LIN {X 0,Y 80.87,Z 798.949,A -85,B 0,C 180,E1 4987.72,E2 4987.72} C_VEL
LIN {X 0,Y 77.511,Z 800.568,A -85,B 0,C 180,E1 4982.778,E2 4982.778} C_VEL
LIN {X 0,Y 74.215,Z 804.27,A -85,B 0,C 180,E1 4966.959,E2 4966.959} C_VEL
LIN {X 0,Y 75.459,Z 805.862,A -85,B 0,C 180,E1 4953.038,E2 4953.038} C_VEL
LIN {X 0,Y 75.99,Z 806.028,A -85,B 0,C 180,E1 4949.467,E2 4949.467} C_VEL
LIN {X 0,Y 74.209,Z 804.782,A -85,B 0,C 180,E1 4936.759,E2 4936.759} C_VEL
LIN {X 0,Y 76.212,Z 801.556,A -85,B 0,C 180,E1 4920.961,E2 4920.961} C_VEL
LIN {X 0,Y 83.236,Z 796.479,A -85,B 0,C 180,E1 4906.789,E2 4906.789} C_VEL
LIN {X 0,Y 94.398,Z 789.488,A -85,B 0,C 180,E1 4895.358,E2 4895.358} C_VEL
LIN {X 0,Y 107.739,Z 780.951,A -85,B 0,C 180,E1 4887.014,E2 4887.014} C_VEL
LIN {X 0,Y 122.056,Z 770.983,A -85,B 0,C 180,E1 4880.958,E2 4880.958} C_VEL
LIN {X 0,Y 136.611,Z 759.652,A -85,B 0,C 180,E1 4876.511,E2 4876.511} C_VEL
LIN {X 0,Y 150.961,Z 747,A -85,B 0,C 180,E1 4873.195,E2 4873.195} C_VEL
LIN {X 0,Y 165.296,Z 732.474,A -85,B 0,C 180,E1 4870.605,E2 4870.605} C_VEL
LIN {X 0,Y 178.339,Z 717.175,A -85,B 0,C 180,E1 4868.706,E2 4868.706} C_VEL
LIN {X 0,Y 190.774,Z 700.081,A -85,B 0,C 180,E1 4867.225,E2 4867.225} C_VEL
LIN {X 0,Y 201.627,Z 682.331,A -85,B 0,C 180,E1 4866.151,E2 4866.151} C_VEL
LIN {X 0,Y 211.381,Z 662.929,A -85,B 0,C 180,E1 4865.337,E2 4865.337} C_VEL
LIN {X 0,Y 219.258,Z 643.158,A -85,B 0,C 180,E1 4864.725,E2 4864.725} C_VEL
LIN {X 0,Y 225.387,Z 622.689,A -85,B 0,C 180,E1 4864.227,E2 4864.227} C_VEL
LIN {X 0,Y 229.672,Z 601.778,A -85,B 0,C 180,E1 4863.811,E2 4863.811} C_VEL
LIN {X 0,Y 238.268,Z 530.43,A -85,B 0,C 180,E1 4862.645,E2 4862.645} C_VEL
LIN {X 0,Y 237.776,Z 527.887,A -85,B 0,C 180,E1 4860.24,E2 4860.24} C_VEL
LIN {X 0,Y 237.596,Z 526.381,A -85,B 0,C 180,E1 4858.07,E2 4858.07} C_VEL
LIN {X 0,Y 237.865,Z 526.25,A -85,B 0,C 180,E1 4853.967,E2 4853.967} C_VEL
LIN {X 0,Y 238.211,Z 526.899,A -85,B 0,C 180,E1 4852.402,E2 4852.402} C_VEL
LIN {X 0,Y 238.456,Z 528.071,A -85,B 0,C 180,E1 4851.324,E2 4851.324} C_VEL
LIN {X 0,Y 231.321,Z 589.425,A -85,B 0,C 180,E1 4850.247,E2 4850.247} C_VEL
LIN {X 0,Y 228.042,Z 608.919,A -85,B 0,C 180,E1 4849.701,E2 4849.701} C_VEL
LIN {X 0,Y 223.305,Z 627.563,A -85,B 0,C 180,E1 4849.015,E2 4849.015} C_VEL
LIN {X 0,Y 217.088,Z 645.659,A -85,B 0,C 180,E1 4848.153,E2 4848.153} C_VEL
LIN {X 0,Y 208.731,Z 664.585,A -85,B 0,C 180,E1 4846.988,E2 4846.988} C_VEL
LIN {X 0,Y 198.839,Z 682.549,A -85,B 0,C 180,E1 4845.556,E2 4845.556} C_VEL
LIN {X 0,Y 187.897,Z 698.953,A -85,B 0,C 180,E1 4843.836,E2 4843.836} C_VEL
LIN {X 0,Y 175.842,Z 714.135,A -85,B 0,C 180,E1 4841.724,E2 4841.724} C_VEL
LIN {X 0,Y 162.701,Z 728.173,A -85,B 0,C 180,E1 4839.079,E2 4839.079} C_VEL
LIN {X 0,Y 149.063,Z 740.606,A -85,B 0,C 180,E1 4835.812,E2 4835.812} C_VEL
LIN {X 0,Y 135.111,Z 751.51,A -85,B 0,C 180,E1 4831.716,E2 4831.716} C_VEL
LIN {X 0,Y 120.926,Z 761.042,A -85,B 0,C 180,E1 4826.358,E2 4826.358} C_VEL
LIN {X 0,Y 107.001,Z 769.093,A -85,B 0,C 180,E1 4819.19,E2 4819.19} C_VEL
LIN {X 0,Y 94.79,Z 775.203,A -85,B 0,C 180,E1 4810.047,E2 4810.047} C_VEL
LIN {X 0,Y 85.286,Z 779.428,A -85,B 0,C 180,E1 4798.728,E2 4798.728} C_VEL
LIN {X 0,Y 79.196,Z 781.917,A -85,B 0,C 180,E1 4785.374,E2 4785.374} C_VEL
LIN {X 0,Y 77.022,Z 782.778,A -85,B 0,C 180,E1 4770.744,E2 4770.744} C_VEL
LIN {X 0,Y 78.595,Z 782.144,A -85,B 0,C 180,E1 4756.763,E2 4756.763} C_VEL
LIN {X 0,Y 84.097,Z 779.929,A -85,B 0,C 180,E1 4743.142,E2 4743.142} C_VEL
LIN {X 0,Y 93.116,Z 776.003,A -85,B 0,C 180,E1 4731.481,E2 4731.481} C_VEL
LIN {X 0,Y 104.314,Z 770.552,A -85,B 0,C 180,E1 4722.436,E2 4722.436} C_VEL
LIN {X 0,Y 117.401,Z 763.276,A -85,B 0,C 180,E1 4715.158,E2 4715.158} C_VEL
LIN {X 0,Y 131.069,Z 754.49,A -85,B 0,C 180,E1 4709.586,E2 4709.586} C_VEL
LIN {X 0,Y 145.656,Z 743.569,A -85,B 0,C 180,E1 4705.03,E2 4705.03} C_VEL
LIN {X 0,Y 159.184,Z 731.747,A -85,B 0,C 180,E1 4701.631,E2 4701.631} C_VEL
LIN {X 0,Y 172.242,Z 718.44,A -85,B 0,C 180,E1 4698.884,E2 4698.884} C_VEL
LIN {X 0,Y 184.101,Z 704.311,A -85,B 0,C 180,E1 4696.73,E2 4696.73} C_VEL
LIN {X 0,Y 195.07,Z 688.928,A -85,B 0,C 180,E1 4694.95,E2 4694.95} C_VEL
LIN {X 0,Y 205.1,Z 672.108,A -85,B 0,C 180,E1 4693.461,E2 4693.461} C_VEL
LIN {X 0,Y 213.82,Z 654.238,A -85,B 0,C 180,E1 4692.234,E2 4692.234} C_VEL
LIN {X 0,Y 220.959,Z 635.839,A -85,B 0,C 180,E1 4691.251,E2 4691.251} C_VEL
LIN {X 0,Y 226.74,Z 615.995,A -85,B 0,C 180,E1 4690.436,E2 4690.436} C_VEL
LIN {X 0,Y 230.757,Z 595.786,A -85,B 0,C 180,E1 4689.81,E2 4689.81} C_VEL
LIN {X 0,Y 236.026,Z 551.57,A -85,B 0,C 180,E1 4688.94,E2 4688.94} C_VEL
LIN {X 0,Y 238.75,Z 528.075,A -85,B 0,C 180,E1 4688.563,E2 4688.563} C_VEL
LIN {X 0,Y 238.273,Z 526.572,A -85,B 0,C 180,E1 4686.506,E2 4686.506} C_VEL
LIN {X 0,Y 237.888,Z 526.562,A -85,B 0,C 180,E1 4682.168,E2 4682.168} C_VEL
LIN {X 0,Y 238.215,Z 528.774,A -85,B 0,C 180,E1 4678.918,E2 4678.918} C_VEL
LIN {X 0,Y 238.522,Z 530.833,A -85,B 0,C 180,E1 4677.356,E2 4677.356} C_VEL
LIN {X 0,Y 229.693,Z 603.415,A -85,B 0,C 180,E1 4676.168,E2 4676.168} C_VEL
LIN {X 0,Y 225.268,Z 624.242,A -85,B 0,C 180,E1 4675.75,E2 4675.75} C_VEL
LIN {X 0,Y 219.212,Z 644.095,A -85,B 0,C 180,E1 4675.261,E2 4675.261} C_VEL
LIN {X 0,Y 211.383,Z 663.553,A -85,B 0,C 180,E1 4674.655,E2 4674.655} C_VEL
LIN {X 0,Y 202.115,Z 681.945,A -85,B 0,C 180,E1 4673.885,E2 4673.885} C_VEL
LIN {X 0,Y 190.896,Z 700.299,A -85,B 0,C 180,E1 4672.779,E2 4672.779} C_VEL
LIN {X 0,Y 178.447,Z 717.368,A -85,B 0,C 180,E1 4671.299,E2 4671.299} C_VEL
LIN {X 0,Y 164.832,Z 733.27,A -85,B 0,C 180,E1 4669.311,E2 4669.311} C_VEL
LIN {X 0,Y 150.054,Z 748.089,A -85,B 0,C 180,E1 4666.61,E2 4666.61} C_VEL
LIN {X 0,Y 134.86,Z 761.302,A -85,B 0,C 180,E1 4663.016,E2 4663.016} C_VEL
LIN {X 0,Y 119.586,Z 772.97,A -85,B 0,C 180,E1 4658.131,E2 4658.131} C_VEL
LIN {X 0,Y 104.755,Z 783.066,A -85,B 0,C 180,E1 4651.412,E2 4651.412} C_VEL
LIN {X 0,Y 91.293,Z 791.543,A -85,B 0,C 180,E1 4642.049,E2 4642.049} C_VEL
LIN {X 0,Y 81.046,Z 798.03,A -85,B 0,C 180,E1 4629.904,E2 4629.904} C_VEL
LIN {X 0,Y 77.511,Z 800.568,A -85,B 0,C 180,E1 4622.778,E2 4622.778} C_VEL
LIN {X 0,Y 74.757,Z 801.989,A -85,B 0,C 180,E1 4617.407,E2 4617.407} C_VEL
LIN {X 0,Y 68.448,Z 803.712,A -85,B 0,C 180,E1 4605.965,E2 4605.965} C_VEL
LIN {X 0,Y 66.797,Z 804.343,A -85,B 0,C 180,E1 4598.037,E2 4598.037} C_VEL
LIN {X 0,Y 66.981,Z 804.481,A -85,B 0,C 180,E1 4595.654,E2 4595.654} C_VEL
LIN {X 0,Y 67.99,Z 804.819,A -85,B 0,C 180,E1 4589.63,E2 4589.63} C_VEL
LIN {X 0,Y 66.248,Z 803.424,A -85,B 0,C 180,E1 4574.237,E2 4574.237} C_VEL
LIN {X 0,Y 69.077,Z 800.295,A -85,B 0,C 180,E1 4557.619,E2 4557.619} C_VEL
LIN {X 0,Y 77.372,Z 795.212,A -85,B 0,C 180,E1 4542.559,E2 4542.559} C_VEL
LIN {X 0,Y 89.824,Z 788.216,A -85,B 0,C 180,E1 4531.009,E2 4531.009} C_VEL
LIN {X 0,Y 104.215,Z 779.674,A -85,B 0,C 180,E1 4522.924,E2 4522.924} C_VEL
LIN {X 0,Y 119.332,Z 769.699,A -85,B 0,C 180,E1 4517.223,E2 4517.223} C_VEL
LIN {X 0,Y 134.489,Z 758.36,A -85,B 0,C 180,E1 4513.12,E2 4513.12} C_VEL
LIN {X 0,Y 149.29,Z 745.693,A -85,B 0,C 180,E1 4510.102,E2 4510.102} C_VEL
LIN {X 0,Y 163.502,Z 731.675,A -85,B 0,C 180,E1 4507.843,E2 4507.843} C_VEL
LIN {X 0,Y 176.979,Z 716.205,A -85,B 0,C 180,E1 4506.12,E2 4506.12} C_VEL
LIN {X 0,Y 189.635,Z 699.109,A -85,B 0,C 180,E1 4504.808,E2 4504.808} C_VEL
LIN {X 0,Y 200.918,Z 680.865,A -85,B 0,C 180,E1 4503.846,E2 4503.846} C_VEL
LIN {X 0,Y 210.287,Z 662.45,A -85,B 0,C 180,E1 4503.175,E2 4503.175} C_VEL
LIN {X 0,Y 218.195,Z 642.955,A -85,B 0,C 180,E1 4502.643,E2 4502.643} C_VEL
LIN {X 0,Y 224.532,Z 622.209,A -85,B 0,C 180,E1 4502.192,E2 4502.192} C_VEL
LIN {X 0,Y 228.935,Z 601.111,A -85,B 0,C 180,E1 4501.809,E2 4501.809} C_VEL
LIN {X 0,Y 236.861,Z 536.432,A -85,B 0,C 180,E1 4500.801,E2 4500.801} C_VEL
LIN {X 0,Y 236.592,Z 534.278,A -85,B 0,C 180,E1 4497.82,E2 4497.82} C_VEL
LIN {X 0,Y 236.945,Z 534.241,A -85,B 0,C 180,E1 4493.701,E2 4493.701} C_VEL
LIN {X 0,Y 237.048,Z 534.547,A -85,B 0,C 180,E1 4493.152,E2 4493.152} C_VEL
LIN {X 0,Y 230.283,Z 591.262,A -85,B 0,C 180,E1 4492.187,E2 4492.187} C_VEL
LIN {X 0,Y 226.761,Z 611.086,A -85,B 0,C 180,E1 4491.649,E2 4491.649} C_VEL
LIN {X 0,Y 221.706,Z 630.042,A -85,B 0,C 180,E1 4490.977,E2 4490.977} C_VEL
LIN {X 0,Y 215.141,Z 648.362,A -85,B 0,C 180,E1 4490.141,E2 4490.141} C_VEL
LIN {X 0,Y 206.72,Z 666.747,A -85,B 0,C 180,E1 4489.064,E2 4489.064} C_VEL
LIN {X 0,Y 196.939,Z 684.033,A -85,B 0,C 180,E1 4487.766,E2 4487.766} C_VEL
LIN {X 0,Y 185.854,Z 700.262,A -85,B 0,C 180,E1 4486.174,E2 4486.174} C_VEL
LIN {X 0,Y 173.527,Z 715.411,A -85,B 0,C 180,E1 4484.201,E2 4484.201} C_VEL
LIN {X 0,Y 160.047,Z 729.424,A -85,B 0,C 180,E1 4481.724,E2 4481.724} C_VEL
LIN {X 0,Y 145.999,Z 741.842,A -85,B 0,C 180,E1 4478.647,E2 4478.647} C_VEL
LIN {X 0,Y 131.542,Z 752.736,A -85,B 0,C 180,E1 4474.756,E2 4474.756} C_VEL
LIN {X 0,Y 116.962,Z 762.108,A -85,B 0,C 180,E1 4469.699,E2 4469.699} C_VEL
LIN {X 0,Y 102.702,Z 769.932,A -85,B 0,C 180,E1 4462.967,E2 4462.967} C_VEL
LIN {X 0,Y 89.463,Z 776.145,A -85,B 0,C 180,E1 4453.861,E2 4453.861} C_VEL
LIN {X 0,Y 78.868,Z 780.452,A -85,B 0,C 180,E1 4442.171,E2 4442.171} C_VEL
LIN {X 0,Y 71.832,Z 783.018,A -85,B 0,C 180,E1 4427.832,E2 4427.832} C_VEL
LIN {X 0,Y 69.156,Z 783.937,A -85,B 0,C 180,E1 4412.486,E2 4412.486} C_VEL
LIN {X 0,Y 70.527,Z 783.466,A -85,B 0,C 180,E1 4396.89,E2 4396.89} C_VEL
LIN {X 0,Y 76.303,Z 781.422,A -85,B 0,C 180,E1 4381.854,E2 4381.854} C_VEL
LIN {X 0,Y 85.91,Z 777.677,A -85,B 0,C 180,E1 4369.328,E2 4369.328} C_VEL
LIN {X 0,Y 98.445,Z 772.088,A -85,B 0,C 180,E1 4359.478,E2 4359.478} C_VEL
LIN {X 0,Y 112.253,Z 764.919,A -85,B 0,C 180,E1 4352.204,E2 4352.204} C_VEL
LIN {X 0,Y 126.523,Z 756.253,A -85,B 0,C 180,E1 4346.752,E2 4346.752} C_VEL
LIN {X 0,Y 140.772,Z 746.14,A -85,B 0,C 180,E1 4342.584,E2 4342.584} C_VEL
LIN {X 0,Y 154.677,Z 734.619,A -85,B 0,C 180,E1 4339.311,E2 4339.311} C_VEL
LIN {X 0,Y 168.049,Z 721.668,A -85,B 0,C 180,E1 4336.687,E2 4336.687} C_VEL
LIN {X 0,Y 180.762,Z 707.191,A -85,B 0,C 180,E1 4334.543,E2 4334.543} C_VEL
LIN {X 0,Y 192.724,Z 690.993,A -85,B 0,C 180,E1 4332.756,E2 4332.756} C_VEL
LIN {X 0,Y 202.946,Z 674.402,A -85,B 0,C 180,E1 4331.366,E2 4331.366} C_VEL
LIN {X 0,Y 211.824,Z 656.824,A -85,B 0,C 180,E1 4330.219,E2 4330.219} C_VEL
LIN {X 0,Y 219.327,Z 638.171,A -85,B 0,C 180,E1 4329.269,E2 4329.269} C_VEL
LIN {X 0,Y 225.338,Z 618.422,A -85,B 0,C 180,E1 4328.491,E2 4328.491} C_VEL
LIN {X 0,Y 229.599,Z 598.14,A -85,B 0,C 180,E1 4327.882,E2 4327.882} C_VEL
LIN {X 0,Y 234.631,Z 557.443,A -85,B 0,C 180,E1 4327.085,E2 4327.085} C_VEL
LIN {X 0,Y 237.333,Z 534.597,A -85,B 0,C 180,E1 4326.714,E2 4326.714} C_VEL
LIN {X 0,Y 236.89,Z 534.461,A -85,B 0,C 180,E1 4322.42,E2 4322.42} C_VEL
LIN {X 0,Y 237.097,Z 536.385,A -85,B 0,C 180,E1 4319.517,E2 4319.517} C_VEL
LIN {X 0,Y 237.127,Z 536.857,A -85,B 0,C 180,E1 4319.187,E2 4319.187} C_VEL
LIN {X 0,Y 228.983,Z 602.568,A -85,B 0,C 180,E1 4318.174,E2 4318.174} C_VEL
LIN {X 0,Y 224.534,Z 623.283,A -85,B 0,C 180,E1 4317.795,E2 4317.795} C_VEL
LIN {X 0,Y 218.444,Z 643.068,A -85,B 0,C 180,E1 4317.363,E2 4317.363} C_VEL
LIN {X 0,Y 210.782,Z 661.997,A -85,B 0,C 180,E1 4316.851,E2 4316.851} C_VEL
LIN {X 0,Y 200.92,Z 681.371,A -85,B 0,C 180,E1 4316.147,E2 4316.147} C_VEL
LIN {X 0,Y 189.637,Z 699.509,A -85,B 0,C 180,E1 4315.184,E2 4315.184} C_VEL
LIN {X 0,Y 176.981,Z 716.533,A -85,B 0,C 180,E1 4313.873,E2 4313.873} C_VEL
LIN {X 0,Y 163.027,Z 732.455,A -85,B 0,C 180,E1 4312.081,E2 4312.081} C_VEL
LIN {X 0,Y 148.356,Z 746.799,A -85,B 0,C 180,E1 4309.72,E2 4309.72} C_VEL
LIN {X 0,Y 132.674,Z 760.024,A -85,B 0,C 180,E1 4306.444,E2 4306.444} C_VEL
LIN {X 0,Y 116.739,Z 771.695,A -85,B 0,C 180,E1 4301.93,E2 4301.93} C_VEL
LIN {X 0,Y 101.029,Z 781.796,A -85,B 0,C 180,E1 4295.571,E2 4295.571} C_VEL
LIN {X 0,Y 86.409,Z 790.275,A -85,B 0,C 180,E1 4286.419,E2 4286.419} C_VEL
LIN {X 0,Y 74.612,Z 796.891,A -85,B 0,C 180,E1 4273.646,E2 4273.646} C_VEL
LIN {X 0,Y 67.665,Z 801.488,A -85,B 0,C 180,E1 4257.556,E2 4257.556} C_VEL
LIN {X 0,Y 66.421,Z 804.095,A -85,B 0,C 180,E1 4240.407,E2 4240.407} C_VEL
LIN {X 0,Y 66.981,Z 804.481,A -85,B 0,C 180,E1 4235.654,E2 4235.654} C_VEL
LIN {X 0,Y 66.693,Z 804.571,A -85,B 0,C 180,E1 4232.598,E2 4232.598} C_VEL
LIN {X 0,Y 64.66,Z 804.284,A -85,B 0,C 180,E1 4228.461,E2 4228.461} C_VEL
LIN {X 0,Y 58.75,Z 802.884,A -85,B 0,C 180,E1 4218.157,E2 4218.157} C_VEL
LIN {X 0,Y 58.309,Z 802.507,A -85,B 0,C 180,E1 4215.107,E2 4215.107} C_VEL
LIN {X 0,Y 61.542,Z 799.446,A -85,B 0,C 180,E1 4195.346,E2 4195.346} C_VEL
LIN {X 0,Y 70.802,Z 794.549,A -85,B 0,C 180,E1 4179.042,E2 4179.042} C_VEL
LIN {X 0,Y 83.558,Z 788.148,A -85,B 0,C 180,E1 4167.692,E2 4167.692} C_VEL
LIN {X 0,Y 99.129,Z 779.667,A -85,B 0,C 180,E1 4159.441,E2 4159.441} C_VEL
LIN {X 0,Y 115.328,Z 769.658,A -85,B 0,C 180,E1 4153.838,E2 4153.838} C_VEL
LIN {X 0,Y 130.975,Z 758.559,A -85,B 0,C 180,E1 4150.019,E2 4150.019} C_VEL
LIN {X 0,Y 147.104,Z 745.276,A -85,B 0,C 180,E1 4147.101,E2 4147.101} C_VEL
LIN {X 0,Y 162.096,Z 730.871,A -85,B 0,C 180,E1 4145.026,E2 4145.026} C_VEL
LIN {X 0,Y 176.293,Z 714.854,A -85,B 0,C 180,E1 4143.469,E2 4143.469} C_VEL
LIN {X 0,Y 189.126,Z 697.707,A -85,B 0,C 180,E1 4142.343,E2 4142.343} C_VEL
LIN {X 0,Y 200.04,Z 680.284,A -85,B 0,C 180,E1 4141.56,E2 4141.56} C_VEL
LIN {X 0,Y 209.496,Z 661.945,A -85,B 0,C 180,E1 4140.993,E2 4140.993} C_VEL
LIN {X 0,Y 217.523,Z 642.437,A -85,B 0,C 180,E1 4140.537,E2 4140.537} C_VEL
LIN {X 0,Y 223.931,Z 621.816,A -85,B 0,C 180,E1 4140.145,E2 4140.145} C_VEL
LIN {X 0,Y 228.431,Z 600.737,A -85,B 0,C 180,E1 4139.801,E2 4139.801} C_VEL
LIN {X 0,Y 235.632,Z 543.029,A -85,B 0,C 180,E1 4138.966,E2 4138.966} C_VEL
LIN {X 0,Y 235.593,Z 542.128,A -85,B 0,C 180,E1 4137.324,E2 4137.324} C_VEL
LIN {X 0,Y 235.733,Z 542.122,A -85,B 0,C 180,E1 4134.985,E2 4134.985} C_VEL
LIN {X 0,Y 229.443,Z 593.572,A -85,B 0,C 180,E1 4134.131,E2 4134.131} C_VEL
LIN {X 0,Y 225.559,Z 614.046,A -85,B 0,C 180,E1 4133.593,E2 4133.593} C_VEL
LIN {X 0,Y 220.134,Z 633.241,A -85,B 0,C 180,E1 4132.937,E2 4132.937} C_VEL
LIN {X 0,Y 212.981,Z 652.126,A -85,B 0,C 180,E1 4132.109,E2 4132.109} C_VEL
LIN {X 0,Y 204.421,Z 669.941,A -85,B 0,C 180,E1 4131.112,E2 4131.112} C_VEL
LIN {X 0,Y 194.523,Z 686.751,A -85,B 0,C 180,E1 4129.916,E2 4129.916} C_VEL
LIN {X 0,Y 183.19,Z 702.748,A -85,B 0,C 180,E1 4128.433,E2 4128.433} C_VEL
LIN {X 0,Y 170.616,Z 717.665,A -85,B 0,C 180,E1 4126.601,E2 4126.601} C_VEL
LIN {X 0,Y 157.746,Z 730.671,A -85,B 0,C 180,E1 4124.453,E2 4124.453} C_VEL
LIN {X 0,Y 143.306,Z 743.076,A -85,B 0,C 180,E1 4121.596,E2 4121.596} C_VEL
LIN {X 0,Y 128.363,Z 753.961,A -85,B 0,C 180,E1 4117.957,E2 4117.957} C_VEL
LIN {X 0,Y 113.169,Z 763.326,A -85,B 0,C 180,E1 4113.166,E2 4113.166} C_VEL
LIN {X 0,Y 97.751,Z 771.333,A -85,B 0,C 180,E1 4106.471,E2 4106.471} C_VEL
LIN {X 0,Y 83.271,Z 777.616,A -85,B 0,C 180,E1 4097.09,E2 4097.09} C_VEL
LIN {X 0,Y 71.46,Z 781.937,A -85,B 0,C 180,E1 4084.355,E2 4084.355} C_VEL
LIN {X 0,Y 63.8,Z 784.403,A -85,B 0,C 180,E1 4068.266,E2 4068.266} C_VEL
LIN {X 0,Y 61.2,Z 785.2,A -85,B 0,C 180,E1 4050,E2 4050} C_VEL
LIN {X 0,Y 63.781,Z 784.429,A -85,B 0,C 180,E1 4031.729,E2 4031.729} C_VEL
LIN {X 0,Y 71.262,Z 782.046,A -85,B 0,C 180,E1 4015.861,E2 4015.861} C_VEL
LIN {X 0,Y 82.576,Z 777.942,A -85,B 0,C 180,E1 4003.408,E2 4003.408} C_VEL
LIN {X 0,Y 95.818,Z 772.302,A -85,B 0,C 180,E1 3994.479,E2 3994.479} C_VEL
LIN {X 0,Y 109.848,Z 765.261,A -85,B 0,C 180,E1 3988.007,E2 3988.007} C_VEL
LIN {X 0,Y 124.866,Z 756.375,A -85,B 0,C 180,E1 3982.952,E2 3982.952} C_VEL
LIN {X 0,Y 139.694,Z 746.022,A -85,B 0,C 180,E1 3979.133,E2 3979.133} C_VEL
LIN {X 0,Y 154.055,Z 734.233,A -85,B 0,C 180,E1 3976.152,E2 3976.152} C_VEL
LIN {X 0,Y 167.795,Z 720.972,A -85,B 0,C 180,E1 3973.77,E2 3973.77} C_VEL
LIN {X 0,Y 180.342,Z 706.72,A -85,B 0,C 180,E1 3971.895,E2 3971.895} C_VEL
LIN {X 0,Y 191.484,Z 691.818,A -85,B 0,C 180,E1 3970.405,E2 3970.405} C_VEL
LIN {X 0,Y 201.999,Z 674.988,A -85,B 0,C 180,E1 3969.114,E2 3969.114} C_VEL
LIN {X 0,Y 211.047,Z 657.306,A -85,B 0,C 180,E1 3968.057,E2 3968.057} C_VEL
LIN {X 0,Y 218.915,Z 637.859,A -85,B 0,C 180,E1 3967.149,E2 3967.149} C_VEL
LIN {X 0,Y 224.94,Z 617.986,A -85,B 0,C 180,E1 3966.432,E2 3966.432} C_VEL
LIN {X 0,Y 229.184,Z 597.547,A -85,B 0,C 180,E1 3965.866,E2 3965.866} C_VEL
LIN {X 0,Y 234.66,Z 553.561,A -85,B 0,C 180,E1 3965.077,E2 3965.077} C_VEL
LIN {X 0,Y 236.022,Z 542.248,A -85,B 0,C 180,E1 3964.901,E2 3964.901} C_VEL
LIN {X 0,Y 235.911,Z 542.576,A -85,B 0,C 180,E1 3961.944,E2 3961.944} C_VEL
LIN {X 0,Y 235.906,Z 543.467,A -85,B 0,C 180,E1 3961.03,E2 3961.03} C_VEL
LIN {X 0,Y 228.524,Z 601.888,A -85,B 0,C 180,E1 3960.186,E2 3960.186} C_VEL
LIN {X 0,Y 224.052,Z 622.449,A -85,B 0,C 180,E1 3959.849,E2 3959.849} C_VEL
LIN {X 0,Y 217.921,Z 642.174,A -85,B 0,C 180,E1 3959.475,E2 3959.475} C_VEL
LIN {X 0,Y 209.994,Z 661.529,A -85,B 0,C 180,E1 3959.027,E2 3959.027} C_VEL
LIN {X 0,Y 200.538,Z 679.92,A -85,B 0,C 180,E1 3958.464,E2 3958.464} C_VEL
LIN {X 0,Y 189.127,Z 698.131,A -85,B 0,C 180,E1 3957.649,E2 3957.649} C_VEL
LIN {X 0,Y 176.294,Z 715.199,A -85,B 0,C 180,E1 3956.523,E2 3956.523} C_VEL
LIN {X 0,Y 162.585,Z 730.642,A -85,B 0,C 180,E1 3955.025,E2 3955.025} C_VEL
LIN {X 0,Y 147.106,Z 745.507,A -85,B 0,C 180,E1 3952.891,E2 3952.891} C_VEL
LIN {X 0,Y 130.978,Z 758.744,A -85,B 0,C 180,E1 3949.975,E2 3949.975} C_VEL
LIN {X 0,Y 114.43,Z 770.421,A -85,B 0,C 180,E1 3945.897,E2 3945.897} C_VEL
LIN {X 0,Y 97.874,Z 780.525,A -85,B 0,C 180,E1 3940.022,E2 3940.022} C_VEL
LIN {X 0,Y 82.085,Z 789.006,A -85,B 0,C 180,E1 3931.282,E2 3931.282} C_VEL
LIN {X 0,Y 69.092,Z 795.5,A -85,B 0,C 180,E1 3918.806,E2 3918.806} C_VEL
LIN {X 0,Y 60.631,Z 800.105,A -85,B 0,C 180,E1 3901.849,E2 3901.849} C_VEL
LIN {X 0,Y 58.387,Z 802.851,A -85,B 0,C 180,E1 3881.858,E2 3881.858} C_VEL
LIN {X 0,Y 59.99,Z 803.61,A -85,B 0,C 180,E1 3869.92,E2 3869.92} C_VEL
LIN {X 0,Y 58.309,Z 802.507,A -85,B 0,C 180,E1 3855.107,E2 3855.107} C_VEL
LIN {X 0,Y 57.755,Z 801.514,A -85,B 0,C 180,E1 3847.524,E2 3847.524} C_VEL
LIN {X 0,Y 57.592,Z 797.296,A -85,B 0,C 180,E1 3826.102,E2 3826.102} C_VEL
LIN {X 0,Y 59.976,Z 795.854,A -85,B 0,C 180,E1 3820.775,E2 3820.775} C_VEL
LIN {X 0,Y 72.988,Z 790.122,A -85,B 0,C 180,E1 3807.075,E2 3807.075} C_VEL
LIN {X 0,Y 88.363,Z 782.767,A -85,B 0,C 180,E1 3798.11,E2 3798.11} C_VEL
LIN {X 0,Y 104.879,Z 773.742,A -85,B 0,C 180,E1 3792.106,E2 3792.106} C_VEL
LIN {X 0,Y 121.175,Z 763.407,A -85,B 0,C 180,E1 3788.053,E2 3788.053} C_VEL
LIN {X 0,Y 137.53,Z 751.311,A -85,B 0,C 180,E1 3785.139,E2 3785.139} C_VEL
LIN {X 0,Y 153.668,Z 737.323,A -85,B 0,C 180,E1 3782.983,E2 3782.983} C_VEL
LIN {X 0,Y 168.442,Z 722.251,A -85,B 0,C 180,E1 3781.454,E2 3781.454} C_VEL
LIN {X 0,Y 181.972,Z 705.964,A -85,B 0,C 180,E1 3780.349,E2 3780.349} C_VEL
LIN {X 0,Y 193.973,Z 688.764,A -85,B 0,C 180,E1 3779.563,E2 3779.563} C_VEL
LIN {X 0,Y 204.496,Z 670.555,A -85,B 0,C 180,E1 3779.006,E2 3779.006} C_VEL
LIN {X 0,Y 213.528,Z 651.227,A -85,B 0,C 180,E1 3778.59,E2 3778.59} C_VEL
LIN {X 0,Y 220.816,Z 631.121,A -85,B 0,C 180,E1 3778.242,E2 3778.242} C_VEL
LIN {X 0,Y 226.297,Z 610.268,A -85,B 0,C 180,E1 3777.927,E2 3777.927} C_VEL
LIN {X 0,Y 229.862,Z 588.948,A -85,B 0,C 180,E1 3777.629,E2 3777.629} C_VEL
LIN {X 0,Y 234.62,Z 550.029,A -85,B 0,C 180,E1 3777.068,E2 3777.068} C_VEL
LIN {X 0,Y 234.603,Z 550.172,A -85,B 0,C 180,E1 3776.831,E2 3776.831} C_VEL
LIN {X 0,Y 228.774,Z 596.534,A -85,B 0,C 180,E1 3776.072,E2 3776.072} C_VEL
LIN {X 0,Y 224.789,Z 616.292,A -85,B 0,C 180,E1 3775.574,E2 3775.574} C_VEL
LIN {X 0,Y 219.306,Z 634.998,A -85,B 0,C 180,E1 3774.974,E2 3774.974} C_VEL
LIN {X 0,Y 212.044,Z 653.683,A -85,B 0,C 180,E1 3774.214,E2 3774.214} C_VEL
LIN {X 0,Y 202.871,Z 672.256,A -85,B 0,C 180,E1 3773.253,E2 3773.253} C_VEL
LIN {X 0,Y 192.291,Z 689.613,A -85,B 0,C 180,E1 3772.104,E2 3772.104} C_VEL
LIN {X 0,Y 180.343,Z 705.825,A -85,B 0,C 180,E1 3770.695,E2 3770.695} C_VEL
LIN {X 0,Y 167.071,Z 720.899,A -85,B 0,C 180,E1 3768.948,E2 3768.948} C_VEL
LIN {X 0,Y 152.678,Z 734.658,A -85,B 0,C 180,E1 3766.749,E2 3766.749} C_VEL
LIN {X 0,Y 137.345,Z 747.003,A -85,B 0,C 180,E1 3763.929,E2 3763.929} C_VEL
LIN {X 0,Y 121.154,Z 757.938,A -85,B 0,C 180,E1 3760.185,E2 3760.185} C_VEL
LIN {X 0,Y 105.121,Z 766.97,A -85,B 0,C 180,E1 3755.258,E2 3755.258} C_VEL
LIN {X 0,Y 89.249,Z 774.383,A -85,B 0,C 180,E1 3748.365,E2 3748.365} C_VEL
LIN {X 0,Y 74.638,Z 780.002,A -85,B 0,C 180,E1 3738.604,E2 3738.604} C_VEL
LIN {X 0,Y 62.804,Z 783.772,A -85,B 0,C 180,E1 3724.968,E2 3724.968} C_VEL
LIN {X 0,Y 55.242,Z 785.846,A -85,B 0,C 180,E1 3706.833,E2 3706.833} C_VEL
LIN {X 0,Y 53.351,Z 786.348,A -85,B 0,C 180,E1 3686.777,E2 3686.777} C_VEL
LIN {X 0,Y 56.942,Z 785.467,A -85,B 0,C 180,E1 3667.276,E2 3667.276} C_VEL
LIN {X 0,Y 65.952,Z 782.941,A -85,B 0,C 180,E1 3650.453,E2 3650.453} C_VEL
LIN {X 0,Y 78.749,Z 778.667,A -85,B 0,C 180,E1 3638.078,E2 3638.078} C_VEL
LIN {X 0,Y 93.957,Z 772.498,A -85,B 0,C 180,E1 3629.24,E2 3629.24} C_VEL
LIN {X 0,Y 109.988,Z 764.604,A -85,B 0,C 180,E1 3623.011,E2 3623.011} C_VEL
LIN {X 0,Y 126.173,Z 754.999,A -85,B 0,C 180,E1 3618.481,E2 3618.481} C_VEL
LIN {X 0,Y 141.882,Z 743.858,A -85,B 0,C 180,E1 3615.11,E2 3615.11} C_VEL
LIN {X 0,Y 156.749,Z 731.349,A -85,B 0,C 180,E1 3612.526,E2 3612.526} C_VEL
LIN {X 0,Y 171.051,Z 717.058,A -85,B 0,C 180,E1 3610.441,E2 3610.441} C_VEL
LIN {X 0,Y 184.125,Z 701.487,A -85,B 0,C 180,E1 3608.778,E2 3608.778} C_VEL
LIN {X 0,Y 195.624,Z 685.09,A -85,B 0,C 180,E1 3607.464,E2 3607.464} C_VEL
LIN {X 0,Y 205.693,Z 667.69,A -85,B 0,C 180,E1 3606.389,E2 3606.389} C_VEL
LIN {X 0,Y 214.444,Z 648.925,A -85,B 0,C 180,E1 3605.481,E2 3605.481} C_VEL
LIN {X 0,Y 221.561,Z 629.164,A -85,B 0,C 180,E1 3604.733,E2 3604.733} C_VEL
LIN {X 0,Y 226.833,Z 608.925,A -85,B 0,C 180,E1 3604.135,E2 3604.135} C_VEL
LIN {X 0,Y 230.244,Z 588.417,A -85,B 0,C 180,E1 3603.668,E2 3603.668} C_VEL
LIN {X 0,Y 234.909,Z 550.241,A -85,B 0,C 180,E1 3603.05,E2 3603.05} C_VEL
LIN {X 0,Y 234.874,Z 550.537,A -85,B 0,C 180,E1 3602.885,E2 3602.885} C_VEL
LIN {X 0,Y 228.383,Z 601.024,A -85,B 0,C 180,E1 3602.206,E2 3602.206} C_VEL
LIN {X 0,Y 223.867,Z 621.585,A -85,B 0,C 180,E1 3601.909,E2 3601.909} C_VEL
LIN {X 0,Y 217.741,Z 641.16,A -85,B 0,C 180,E1 3601.596,E2 3601.596} C_VEL
LIN {X 0,Y 210.013,Z 659.968,A -85,B 0,C 180,E1 3601.24,E2 3601.24} C_VEL
LIN {X 0,Y 200.347,Z 678.704,A -85,B 0,C 180,E1 3600.778,E2 3600.778} C_VEL
LIN {X 0,Y 188.968,Z 696.743,A -85,B 0,C 180,E1 3600.12,E2 3600.12} C_VEL
LIN {X 0,Y 175.988,Z 713.859,A -85,B 0,C 180,E1 3599.186,E2 3599.186} C_VEL
LIN {X 0,Y 161.571,Z 729.855,A -85,B 0,C 180,E1 3597.873,E2 3597.873} C_VEL
LIN {X 0,Y 146.112,Z 744.389,A -85,B 0,C 180,E1 3596.077,E2 3596.077} C_VEL
LIN {X 0,Y 129.791,Z 757.463,A -85,B 0,C 180,E1 3593.583,E2 3593.583} C_VEL
LIN {X 0,Y 112.691,Z 769.146,A -85,B 0,C 180,E1 3590.004,E2 3590.004} C_VEL
LIN {X 0,Y 95.347,Z 779.255,A -85,B 0,C 180,E1 3584.738,E2 3584.738} C_VEL
LIN {X 0,Y 78.415,Z 787.738,A -85,B 0,C 180,E1 3576.64,E2 3576.64} C_VEL
LIN {X 0,Y 63.911,Z 794.235,A -85,B 0,C 180,E1 3564.438,E2 3564.438} C_VEL
LIN {X 0,Y 53.764,Z 798.845,A -85,B 0,C 180,E1 3546.519,E2 3546.519} C_VEL
LIN {X 0,Y 50.391,Z 801.627,A -85,B 0,C 180,E1 3523.538,E2 3523.538} C_VEL
LIN {X 0,Y 51.916,Z 802.384,A -85,B 0,C 180,E1 3510,E2 3510} C_VEL
LIN {X 0,Y 50.587,Z 800.922,A -85,B 0,C 180,E1 3489.16,E2 3489.16} C_VEL
LIN {X 0,Y 56.209,Z 797.564,A -85,B 0,C 180,E1 3467.473,E2 3467.473} C_VEL
LIN {X 0,Y 59.976,Z 795.854,A -85,B 0,C 180,E1 3460.775,E2 3460.775} C_VEL
LIN {X 0,Y 63.488,Z 793.944,A -85,B 0,C 180,E1 3454.597,E2 3454.597} C_VEL
LIN {X 0,Y 73.141,Z 787.653,A -85,B 0,C 180,E1 3439.522,E2 3439.522} C_VEL
LIN {X 0,Y 77.807,Z 785.332,A -85,B 0,C 180,E1 3436.368,E2 3436.368} C_VEL
LIN {X 0,Y 94.429,Z 777.363,A -85,B 0,C 180,E1 3430.037,E2 3430.037} C_VEL
LIN {X 0,Y 111.547,Z 767.711,A -85,B 0,C 180,E1 3425.775,E2 3425.775} C_VEL
LIN {X 0,Y 129.127,Z 755.981,A -85,B 0,C 180,E1 3422.751,E2 3422.751} C_VEL
LIN {X 0,Y 145.985,Z 742.671,A -85,B 0,C 180,E1 3420.653,E2 3420.653} C_VEL
LIN {X 0,Y 161.488,Z 728.226,A -85,B 0,C 180,E1 3419.199,E2 3419.199} C_VEL
LIN {X 0,Y 175.559,Z 712.766,A -85,B 0,C 180,E1 3418.173,E2 3418.173} C_VEL
LIN {X 0,Y 188.154,Z 696.372,A -85,B 0,C 180,E1 3417.452,E2 3417.452} C_VEL
LIN {X 0,Y 199.249,Z 679.077,A -85,B 0,C 180,E1 3416.947,E2 3416.947} C_VEL
LIN {X 0,Y 208.833,Z 660.918,A -85,B 0,C 180,E1 3416.594,E2 3416.594} C_VEL
LIN {X 0,Y 212.676,Z 652.363,A -85,B 0,C 180,E1 3416.453,E2 3416.453} C_VEL
LIN {X 0,Y 204.053,Z 670.181,A -85,B 0,C 180,E1 3415.652,E2 3415.652} C_VEL
LIN {X 0,Y 193.664,Z 687.596,A -85,B 0,C 180,E1 3414.667,E2 3414.667} C_VEL
LIN {X 0,Y 182.141,Z 703.588,A -85,B 0,C 180,E1 3413.496,E2 3413.496} C_VEL
LIN {X 0,Y 169.105,Z 718.73,A -85,B 0,C 180,E1 3412.031,E2 3412.031} C_VEL
LIN {X 0,Y 155.214,Z 732.323,A -85,B 0,C 180,E1 3410.254,E2 3410.254} C_VEL
LIN {X 0,Y 140.061,Z 744.825,A -85,B 0,C 180,E1 3407.954,E2 3407.954} C_VEL
LIN {X 0,Y 124.215,Z 755.806,A -85,B 0,C 180,E1 3404.995,E2 3404.995} C_VEL
LIN {X 0,Y 107.843,Z 765.272,A -85,B 0,C 180,E1 3401.025,E2 3401.025} C_VEL
LIN {X 0,Y 91.236,Z 773.187,A -85,B 0,C 180,E1 3395.447,E2 3395.447} C_VEL
LIN {X 0,Y 75.702,Z 779.207,A -85,B 0,C 180,E1 3387.702,E2 3387.702} C_VEL
LIN {X 0,Y 61.349,Z 783.693,A -85,B 0,C 180,E1 3375.814,E2 3375.814} C_VEL
LIN {X 0,Y 50.55,Z 786.423,A -85,B 0,C 180,E1 3358.34,E2 3358.34} C_VEL
LIN {X 0,Y 45.608,Z 787.501,A -85,B 0,C 180,E1 3336.293,E2 3336.293} C_VEL
LIN {X 0,Y 47.165,Z 787.194,A -85,B 0,C 180,E1 3312.736,E2 3312.736} C_VEL
LIN {X 0,Y 55.349,Z 785.326,A -85,B 0,C 180,E1 3292.108,E2 3292.108} C_VEL
LIN {X 0,Y 67.439,Z 782.004,A -85,B 0,C 180,E1 3278.209,E2 3278.209} C_VEL
LIN {X 0,Y 82.847,Z 776.709,A -85,B 0,C 180,E1 3268.239,E2 3268.239} C_VEL
LIN {X 0,Y 98.957,Z 769.858,A -85,B 0,C 180,E1 3261.638,E2 3261.638} C_VEL
LIN {X 0,Y 115.928,Z 761.002,A -85,B 0,C 180,E1 3256.799,E2 3256.799} C_VEL
LIN {X 0,Y 132.531,Z 750.496,A -85,B 0,C 180,E1 3253.296,E2 3253.296} C_VEL
LIN {X 0,Y 147.58,Z 739.153,A -85,B 0,C 180,E1 3250.78,E2 3250.78} C_VEL
LIN {X 0,Y 162.832,Z 725.464,A -85,B 0,C 180,E1 3248.668,E2 3248.668} C_VEL
LIN {X 0,Y 176.794,Z 710.501,A -85,B 0,C 180,E1 3247.017,E2 3247.017} C_VEL
LIN {X 0,Y 189.401,Z 694.329,A -85,B 0,C 180,E1 3245.691,E2 3245.691} C_VEL
LIN {X 0,Y 200.614,Z 676.933,A -85,B 0,C 180,E1 3244.607,E2 3244.607} C_VEL
LIN {X 0,Y 209.954,Z 659.194,A -85,B 0,C 180,E1 3243.74,E2 3243.74} C_VEL
LIN {X 0,Y 212.304,Z 653.923,A -85,B 0,C 180,E1 3243.519,E2 3243.519} C_VEL
LIN {X 0,Y 203.282,Z 672.394,A -85,B 0,C 180,E1 3243.202,E2 3243.202} C_VEL
LIN {X 0,Y 192.691,Z 690.076,A -85,B 0,C 180,E1 3242.762,E2 3242.762} C_VEL
LIN {X 0,Y 180.67,Z 706.774,A -85,B 0,C 180,E1 3242.133,E2 3242.133} C_VEL
LIN {X 0,Y 167.642,Z 722.073,A -85,B 0,C 180,E1 3241.274,E2 3241.274} C_VEL
LIN {X 0,Y 152.974,Z 736.714,A -85,B 0,C 180,E1 3240.04,E2 3240.04} C_VEL
LIN {X 0,Y 137.036,Z 750.232,A -85,B 0,C 180,E1 3238.303,E2 3238.303} C_VEL
LIN {X 0,Y 120.293,Z 762.301,A -85,B 0,C 180,E1 3235.86,E2 3235.86} C_VEL
LIN {X 0,Y 102.399,Z 773.217,A -85,B 0,C 180,E1 3232.144,E2 3232.144} C_VEL
LIN {X 0,Y 84.326,Z 782.486,A -85,B 0,C 180,E1 3226.471,E2 3226.471} C_VEL
LIN {X 0,Y 67.139,Z 789.96,A -85,B 0,C 180,E1 3217.413,E2 3217.413} C_VEL
LIN {X 0,Y 52.493,Z 795.592,A -85,B 0,C 180,E1 3202.449,E2 3202.449} C_VEL
LIN {X 0,Y 43.546,Z 799.345,A -85,B 0,C 180,E1 3178.827,E2 3178.827} C_VEL
LIN {X 0,Y 43.371,Z 801.043,A -85,B 0,C 180,E1 3152.642,E2 3152.642} C_VEL
LIN {X 0,Y 43.798,Z 801.151,A -85,B 0,C 180,E1 3150,E2 3150} C_VEL
LIN {X 0,Y 42.989,Z 799.656,A -85,B 0,C 180,E1 3125.099,E2 3125.099} C_VEL
LIN {X 0,Y 50.39,Z 796.299,A -85,B 0,C 180,E1 3101.063,E2 3101.063} C_VEL
LIN {X 0,Y 63.995,Z 791.093,A -85,B 0,C 180,E1 3084.949,E2 3084.949} C_VEL
LIN {X 0,Y 77.807,Z 785.332,A -85,B 0,C 180,E1 3076.368,E2 3076.368} C_VEL
LIN {X 0,Y 83.405,Z 782.539,A -85,B 0,C 180,E1 3073.103,E2 3073.103} C_VEL
LIN {X 0,Y 96.694,Z 774.657,A -85,B 0,C 180,E1 3064.844,E2 3064.844} C_VEL
LIN {X 0,Y 102.777,Z 771.132,A -85,B 0,C 180,E1 3062.957,E2 3062.957} C_VEL
LIN {X 0,Y 119.98,Z 760.841,A -85,B 0,C 180,E1 3060.179,E2 3060.179} C_VEL
LIN {X 0,Y 137.042,Z 748.732,A -85,B 0,C 180,E1 3058.227,E2 3058.227} C_VEL
LIN {X 0,Y 153.203,Z 735.16,A -85,B 0,C 180,E1 3056.867,E2 3056.867} C_VEL
LIN {X 0,Y 168.403,Z 720.049,A -85,B 0,C 180,E1 3055.895,E2 3055.895} C_VEL
LIN {X 0,Y 176.106,Z 711.289,A -85,B 0,C 180,E1 3055.477,E2 3055.477} C_VEL
LIN {X 0,Y 161.85,Z 726.387,A -85,B 0,C 180,E1 3054.033,E2 3054.033} C_VEL
LIN {X 0,Y 146.33,Z 740.113,A -85,B 0,C 180,E1 3052.197,E2 3052.197} C_VEL
LIN {X 0,Y 130.009,Z 752.149,A -85,B 0,C 180,E1 3049.86,E2 3049.86} C_VEL
LIN {X 0,Y 112.984,Z 762.559,A -85,B 0,C 180,E1 3046.761,E2 3046.761} C_VEL
LIN {X 0,Y 95.439,Z 771.333,A -85,B 0,C 180,E1 3042.425,E2 3042.425} C_VEL
LIN {X 0,Y 77.711,Z 778.429,A -85,B 0,C 180,E1 3035.992,E2 3035.992} C_VEL
LIN {X 0,Y 61.329,Z 783.568,A -85,B 0,C 180,E1 3026.248,E2 3026.248} C_VEL
LIN {X 0,Y 47.545,Z 786.903,A -85,B 0,C 180,E1 3010.686,E2 3010.686} C_VEL
LIN {X 0,Y 38.855,Z 788.556,A -85,B 0,C 180,E1 2986.443,E2 2986.443} C_VEL
LIN {X 0,Y 38.196,Z 788.652,A -85,B 0,C 180,E1 2957.913,E2 2957.913} C_VEL
LIN {X 0,Y 45.257,Z 787.359,A -85,B 0,C 180,E1 2933.382,E2 2933.382} C_VEL
LIN {X 0,Y 58.267,Z 784.401,A -85,B 0,C 180,E1 2916.246,E2 2916.246} C_VEL
LIN {X 0,Y 74.593,Z 779.556,A -85,B 0,C 180,E1 2905.402,E2 2905.402} C_VEL
LIN {X 0,Y 91.785,Z 773.007,A -85,B 0,C 180,E1 2898.611,E2 2898.611} C_VEL
LIN {X 0,Y 109.214,Z 764.709,A -85,B 0,C 180,E1 2893.974,E2 2893.974} C_VEL
LIN {X 0,Y 126.169,Z 754.817,A -85,B 0,C 180,E1 2890.692,E2 2890.692} C_VEL
LIN {X 0,Y 142.446,Z 743.362,A -85,B 0,C 180,E1 2888.24,E2 2888.24} C_VEL
LIN {X 0,Y 157.935,Z 730.32,A -85,B 0,C 180,E1 2886.328,E2 2886.328} C_VEL
LIN {X 0,Y 172.574,Z 715.584,A -85,B 0,C 180,E1 2884.792,E2 2884.792} C_VEL
LIN {X 0,Y 175.867,Z 711.955,A -85,B 0,C 180,E1 2884.476,E2 2884.476} C_VEL
LIN {X 0,Y 161.304,Z 727.727,A -85,B 0,C 180,E1 2883.673,E2 2883.673} C_VEL
LIN {X 0,Y 145.112,Z 742.471,A -85,B 0,C 180,E1 2882.493,E2 2882.493} C_VEL
LIN {X 0,Y 127.991,Z 755.597,A -85,B 0,C 180,E1 2880.809,E2 2880.809} C_VEL
LIN {X 0,Y 110.028,Z 767.168,A -85,B 0,C 180,E1 2878.333,E2 2878.333} C_VEL
LIN {X 0,Y 91.401,Z 777.171,A -85,B 0,C 180,E1 2874.527,E2 2874.527} C_VEL
LIN {X 0,Y 73.412,Z 785.202,A -85,B 0,C 180,E1 2868.694,E2 2868.694} C_VEL
LIN {X 0,Y 55.883,Z 791.703,A -85,B 0,C 180,E1 2858.489,E2 2858.489} C_VEL
LIN {X 0,Y 41.04,Z 796.501,A -85,B 0,C 180,E1 2839.045,E2 2839.045} C_VEL
LIN {X 0,Y 34.523,Z 799.286,A -85,B 0,C 180,E1 2807.121,E2 2807.121} C_VEL
LIN {X 0,Y 35.661,Z 799.914,A -85,B 0,C 180,E1 2790,E2 2790} C_VEL
LIN {X 0,Y 35.902,Z 798.299,A -85,B 0,C 180,E1 2758.053,E2 2758.053} C_VEL
LIN {X 0,Y 46.034,Z 794.827,A -85,B 0,C 180,E1 2732.107,E2 2732.107} C_VEL
LIN {X 0,Y 61.78,Z 789.533,A -85,B 0,C 180,E1 2717.284,E2 2717.284} C_VEL
LIN {X 0,Y 78.994,Z 782.724,A -85,B 0,C 180,E1 2709.158,E2 2709.158} C_VEL
LIN {X 0,Y 97.233,Z 774.068,A -85,B 0,C 180,E1 2704.101,E2 2704.101} C_VEL
LIN {X 0,Y 102.777,Z 771.132,A -85,B 0,C 180,E1 2702.957,E2 2702.957} C_VEL
LIN {X 0,Y 108.91,Z 767.484,A -85,B 0,C 180,E1 2701.302,E2 2701.302} C_VEL
LIN {X 0,Y 123.429,Z 757.685,A -85,B 0,C 180,E1 2696.388,E2 2696.388} C_VEL
LIN {X 0,Y 129.469,Z 753.349,A -85,B 0,C 180,E1 2695.395,E2 2695.395} C_VEL
LIN {X 0,Y 139.565,Z 745.837,A -85,B 0,C 180,E1 2694.64,E2 2694.64} C_VEL
LIN {X 0,Y 122.874,Z 757.133,A -85,B 0,C 180,E1 2692.518,E2 2692.518} C_VEL
LIN {X 0,Y 105.684,Z 766.726,A -85,B 0,C 180,E1 2689.704,E2 2689.704} C_VEL
LIN {X 0,Y 88.66,Z 774.461,A -85,B 0,C 180,E1 2685.892,E2 2685.892} C_VEL
LIN {X 0,Y 70.329,Z 781.056,A -85,B 0,C 180,E1 2679.766,E2 2679.766} C_VEL
LIN {X 0,Y 53.172,Z 785.723,A -85,B 0,C 180,E1 2669.879,E2 2669.879} C_VEL
LIN {X 0,Y 38.581,Z 788.624,A -85,B 0,C 180,E1 2652.361,E2 2652.361} C_VEL
LIN {X 0,Y 30.097,Z 789.884,A -85,B 0,C 180,E1 2621.498,E2 2621.498} C_VEL
LIN {X 0,Y 32.014,Z 789.659,A -85,B 0,C 180,E1 2586.046,E2 2586.046} C_VEL
LIN {X 0,Y 43.22,Z 787.88,A -85,B 0,C 180,E1 2560.235,E2 2560.235} C_VEL
LIN {X 0,Y 58.957,Z 784.417,A -85,B 0,C 180,E1 2546,E2 2546} C_VEL
LIN {X 0,Y 76.625,Z 779.126,A -85,B 0,C 180,E1 2537.726,E2 2537.726} C_VEL
LIN {X 0,Y 94.268,Z 772.282,A -85,B 0,C 180,E1 2532.637,E2 2532.637} C_VEL
LIN {X 0,Y 112.376,Z 763.438,A -85,B 0,C 180,E1 2529.037,E2 2529.037} C_VEL
LIN {X 0,Y 129.806,Z 752.952,A -85,B 0,C 180,E1 2526.476,E2 2526.476} C_VEL
LIN {X 0,Y 139.027,Z 746.499,A -85,B 0,C 180,E1 2525.314,E2 2525.314} C_VEL
LIN {X 0,Y 122.272,Z 758.394,A -85,B 0,C 180,E1 2523.965,E2 2523.965} C_VEL
LIN {X 0,Y 105.047,Z 768.698,A -85,B 0,C 180,E1 2522.011,E2 2522.011} C_VEL
LIN {X 0,Y 86.005,Z 778.161,A -85,B 0,C 180,E1 2518.764,E2 2518.764} C_VEL
LIN {X 0,Y 67.414,Z 785.69,A -85,B 0,C 180,E1 2513.559,E2 2513.559} C_VEL
LIN {X 0,Y 48.944,Z 791.712,A -85,B 0,C 180,E1 2503.763,E2 2503.763} C_VEL
LIN {X 0,Y 32.862,Z 796.042,A -85,B 0,C 180,E1 2482.282,E2 2482.282} C_VEL
LIN {X 0,Y 26.624,Z 798.324,A -85,B 0,C 180,E1 2442.486,E2 2442.486} C_VEL
LIN {X 0,Y 27.502,Z 798.675,A -85,B 0,C 180,E1 2430,E2 2430} C_VEL
LIN {X 0,Y 29.488,Z 796.969,A -85,B 0,C 180,E1 2388.236,E2 2388.236} C_VEL
LIN {X 0,Y 43.011,Z 793.354,A -85,B 0,C 180,E1 2361.589,E2 2361.589} C_VEL
LIN {X 0,Y 60.769,Z 787.961,A -85,B 0,C 180,E1 2349.182,E2 2349.182} C_VEL
LIN {X 0,Y 79.084,Z 781.053,A -85,B 0,C 180,E1 2342.849,E2 2342.849} C_VEL
LIN {X 0,Y 97.998,Z 772.289,A -85,B 0,C 180,E1 2339.022,E2 2339.022} C_VEL
LIN {X 0,Y 116.181,Z 762.063,A -85,B 0,C 180,E1 2336.634,E2 2336.634} C_VEL
LIN {X 0,Y 129.469,Z 753.349,A -85,B 0,C 180,E1 2335.395,E2 2335.395} C_VEL
LIN {X 0,Y 127.987,Z 754.261,A -85,B 0,C 180,E1 2334.947,E2 2334.947} C_VEL
LIN {X 0,Y 119.86,Z 759.395,A -85,B 0,C 180,E1 2334.356,E2 2334.356} C_VEL
LIN {X 0,Y 103.567,Z 768.51,A -85,B 0,C 180,E1 2334.171,E2 2334.171} C_VEL
LIN {X 0,Y 92.21,Z 774.105,A -85,B 0,C 180,E1 2334.891,E2 2334.891} C_VEL
LIN {X 0,Y 72.025,Z 782.574,A -85,B 0,C 180,E1 2338.157,E2 2338.157} C_VEL
LIN {X 0,Y 51.512,Z 789.275,A -85,B 0,C 180,E1 2344.451,E2 2344.451} C_VEL
LIN {X 0,Y 32.649,Z 793.94,A -85,B 0,C 180,E1 2358.318,E2 2358.318} C_VEL
LIN {X 0,Y 19.334,Z 796.785,A -85,B 0,C 180,E1 2398.859,E2 2398.859} C_VEL
LIN {X 0,Y 19.33,Z 797.434,A -85,B 0,C 180,E1 2429.999,E2 2429.999} C_VEL
LIN {X 0,Y 24.183,Z 795.689,A -85,B 0,C 180,E1 2485.779,E2 2485.779} C_VEL
LIN {X 0,Y 40.689,Z 792.136,A -85,B 0,C 180,E1 2509.387,E2 2509.387} C_VEL
LIN {X 0,Y 60.005,Z 786.763,A -85,B 0,C 180,E1 2518.711,E2 2518.711} C_VEL
LIN {X 0,Y 79.109,Z 779.885,A -85,B 0,C 180,E1 2523.191,E2 2523.191} C_VEL
LIN {X 0,Y 98.515,Z 771.143,A -85,B 0,C 180,E1 2525.826,E2 2525.826} C_VEL
LIN {X 0,Y 102.59,Z 769.098,A -85,B 0,C 180,E1 2526.241,E2 2526.241} C_VEL
LIN {X 0,Y 84.16,Z 776.957,A -85,B 0,C 180,E1 2529.583,E2 2529.583} C_VEL
LIN {X 0,Y 65.164,Z 783.216,A -85,B 0,C 180,E1 2534.846,E2 2534.846} C_VEL
LIN {X 0,Y 47.012,Z 787.573,A -85,B 0,C 180,E1 2543.865,E2 2543.865} C_VEL
LIN {X 0,Y 30.989,Z 790.177,A -85,B 0,C 180,E1 2562.092,E2 2562.092} C_VEL
LIN {X 0,Y 21.979,Z 791.134,A -85,B 0,C 180,E1 2599.516,E2 2599.516} C_VEL
LIN {X 0,Y 26.02,Z 790.716,A -85,B 0,C 180,E1 2645.197,E2 2645.197} C_VEL
LIN {X 0,Y 40.231,Z 788.736,A -85,B 0,C 180,E1 2670.438,E2 2670.438} C_VEL
LIN {X 0,Y 57.781,Z 785.064,A -85,B 0,C 180,E1 2682.122,E2 2682.122} C_VEL
LIN {X 0,Y 75.563,Z 779.885,A -85,B 0,C 180,E1 2688.28,E2 2688.28} C_VEL
LIN {X 0,Y 93.841,Z 772.906,A -85,B 0,C 180,E1 2692.253,E2 2692.253} C_VEL
LIN {X 0,Y 102.592,Z 768.942,A -85,B 0,C 180,E1 2693.754,E2 2693.754} C_VEL
LIN {X 0,Y 92.21,Z 774.105,A -85,B 0,C 180,E1 2694.891,E2 2694.891} C_VEL
LIN {X 0,Y 84.152,Z 777.602,A -85,B 0,C 180,E1 2695.308,E2 2695.308} C_VEL
LIN {X 0,Y 73.515,Z 781.417,A -85,B 0,C 180,E1 2694.359,E2 2694.359} C_VEL
LIN {X 0,Y 55.026,Z 786.476,A -85,B 0,C 180,E1 2689.629,E2 2689.629} C_VEL
LIN {X 0,Y 54.43,Z 786.622,A -85,B 0,C 180,E1 2689.434,E2 2689.434} C_VEL
LIN {X 0,Y 36.055,Z 790.087,A -85,B 0,C 180,E1 2680.537,E2 2680.537} C_VEL
LIN {X 0,Y 19.375,Z 791.979,A -85,B 0,C 180,E1 2656.259,E2 2656.259} C_VEL
LIN {X 0,Y 14.568,Z 792.315,A -85,B 0,C 180,E1 2589.932,E2 2589.932} C_VEL
LIN {X 0,Y 28.04,Z 791.175,A -85,B 0,C 180,E1 2546.946,E2 2546.946} C_VEL
LIN {X 0,Y 46.287,Z 788.398,A -85,B 0,C 180,E1 2533.582,E2 2533.582} C_VEL
LIN {X 0,Y 65.449,Z 783.885,A -85,B 0,C 180,E1 2527.462,E2 2527.462} C_VEL
LIN {X 0,Y 45.055,Z 789.688,A -85,B 0,C 180,E1 2523.031,E2 2523.031} C_VEL
LIN {X 0,Y 25.282,Z 793.681,A -85,B 0,C 180,E1 2511.374,E2 2511.374} C_VEL
LIN {X 0,Y 10.957,Z 795.875,A -85,B 0,C 180,E1 2457.146,E2 2457.146} C_VEL
LIN {X 0,Y 11.138,Z 796.189,A -85,B 0,C 180,E1 2429.999,E2 2429.999} C_VEL
LIN {X 0,Y 20.688,Z 794.409,A -85,B 0,C 180,E1 2354.854,E2 2354.854} C_VEL
LIN {X 0,Y 41.009,Z 790.615,A -85,B 0,C 180,E1 2338.387,E2 2338.387} C_VEL
LIN {X 0,Y 61.427,Z 785.12,A -85,B 0,C 180,E1 2333.161,E2 2333.161} C_VEL
LIN {X 0,Y 65.554,Z 783.757,A -85,B 0,C 180,E1 2332.476,E2 2332.476} C_VEL
LIN {X 0,Y 54.43,Z 786.622,A -85,B 0,C 180,E1 2329.434,E2 2329.434} C_VEL
LIN {X 0,Y 45.975,Z 788.577,A -85,B 0,C 180,E1 2327.472,E2 2327.472} C_VEL
LIN {X 0,Y 29.71,Z 791.568,A -85,B 0,C 180,E1 2326.261,E2 2326.261} C_VEL
LIN {X 0,Y 18.429,Z 792.943,A -85,B 0,C 180,E1 2322.637,E2 2322.637} C_VEL
LIN {X 0,Y 14.841,Z 793.195,A -85,B 0,C 180,E1 2318.285,E2 2318.285} C_VEL
LIN {X 0,Y 7.637,Z 793.517,A -85,B 0,C 180,E1 2209.115,E2 2209.115} C_VEL
LIN {X 0,Y 25.449,Z 792.378,A -85,B 0,C 180,E1 2170.836,E2 2170.836} C_VEL
LIN {X 0,Y 25.834,Z 792.351,A -85,B 0,C 180,E1 2170.381,E2 2170.381} C_VEL
LIN {X 0,Y 5.219,Z 794.622,A -85,B 0,C 180,E1 2143.293,E2 2143.293} C_VEL
LIN {X 0,Y 2.926,Z 794.942,A -85,B 0,C 180,E1 2069.996,E2 2069.996} C_VEL
LIN {X 0,Y 20.232,Z 793.147,A -85,B 0,C 180,E1 1971.468,E2 1971.468} C_VEL
LIN {X 0,Y 26.162,Z 792.265,A -85,B 0,C 180,E1 1969.529,E2 1969.529} C_VEL
LIN {X 0,Y 14.841,Z 793.195,A -85,B 0,C 180,E1 1958.285,E2 1958.285} C_VEL
LIN {X 0,Y 13.153,Z 795.191,A -85,B 0,C 180,E1 1954.913,E2 1954.913} C_VEL
LIN {X 0,Y 13.153,Z 875,A -85,B 0,C 180,E1 1954.913,E2 1954.913} C_VEL
LIN {X 0,Y 13.153,Z 875,A -85,B 0,C 180,E1 1954.913,E2 1954.913}

QRS_NEXT_CUT()

QRS_NEXT()
QRS_HOME()

END
